// TIA Portal project "TemporizadorTON" (V16)

(* hardware
DEVICE "S7-1200 station_1"  S7-1200 Station
   slot 0: "Rack_0"  S7-1200 Rack  Rack  V1.0
   slot 1: "PLC_1"  CPU 1214C AC/DC/Rly  6ES7 214-1BG40-0XB0  V4.4
*)

// ===== PLC "PLC_1"  CPU 1214C AC/DC/Rly =====

VAR_GLOBAL   // PLC tag table "Tabla de variables estándar"
   "Tag_1" AT %I0.0 : Bool;
   "Tag_2" AT %MD100 : Time;
   "Tag_3" AT %Q0.0 : Bool;
   "Tag_4" AT %I0.1 : Bool;
   "Tag_5" AT %MD101 : Time;
   "Tag_6" AT %Q0.1 : Bool;
   "MEMORIA" AT %MD102 : Time;
   "PULSADOR" AT %I0.2 : Bool;
   "RESET" AT %I0.3 : Bool;
END_VAR

// folder: System blocks/Program resources

DATA_BLOCK "IEC_Timer_0_DB"   // DB1
{ S7_Optimized_Access := 'TRUE' }
AUTHOR : Simatic
FAMILY : IEC
NAME : IEC_TMR
VERSION : 1.0
// stored: InstanceOfName IEC_TIMER
"IEC_TIMER"
BEGIN
END_DATA_BLOCK

DATA_BLOCK "IEC_Timer_0_DB_1"   // DB2
{ S7_Optimized_Access := 'TRUE' }
AUTHOR : Simatic
FAMILY : IEC
NAME : IEC_TMR
VERSION : 1.0
// stored: InstanceOfName IEC_TIMER
"IEC_TIMER"
BEGIN
END_DATA_BLOCK

DATA_BLOCK "IEC_Timer_0_DB_2"   // DB3
{ S7_Optimized_Access := 'TRUE' }
AUTHOR : Simatic
FAMILY : IEC
NAME : IEC_TMR
VERSION : 1.0
// stored: InstanceOfName IEC_TIMER
"IEC_TIMER"
BEGIN
END_DATA_BLOCK

// folder: (top level)

ORGANIZATION_BLOCK "Main"   // OB1, LAD, ProgramCycle
TITLE = "Main Program Sweep (Cycle)"
{ S7_Optimized_Access := 'TRUE' }
VERSION : 0.1
// Funcionamiento de TON. También conocido como "Retardo a la conexión"
   VAR_INPUT
      Initial_Call : Bool;   // Initial call of this OB
      Remanence : Bool;   // =True, if remanent data are available
   END_VAR
BEGIN

REGION Network 1
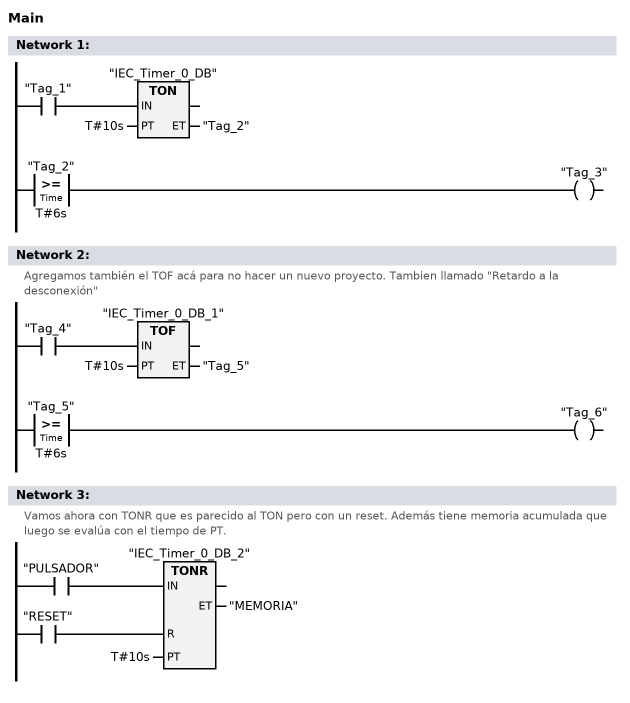
   "IEC_Timer_0_DB".TON(IN := "Tag_1", PT := T#10s, ET => "Tag_2");
   "Tag_3" := "Tag_2" >= T#6s;
END_REGION

REGION Network 2
   // Agregamos también el TOF acá para no hacer un nuevo proyecto. Tambien llamado "Retardo a la desconexión"
   "IEC_Timer_0_DB_1".TOF(IN := "Tag_4", PT := T#10s, ET => "Tag_5");
   "Tag_6" := "Tag_5" >= T#6s;
END_REGION

REGION Network 3
   // Vamos ahora con TONR que es parecido al TON pero con un reset. Además tiene memoria acumulada que luego se evalúa con el tiempo de PT.
   "IEC_Timer_0_DB_2".TONR(IN := "PULSADOR", R := "RESET", PT := T#10s, ET => "MEMORIA");
END_REGION
END_ORGANIZATION_BLOCK